FUNCTION_BLOCK F_UINT_TO_LINT (* convert UINT to LINT *)
  (* Standard: 61131-3; Classification: type conversion function *)
  (* Version 0.0, 2011-12-25, 4DIAC-IDE, 4DIAC-Consortium *)
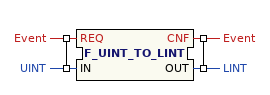
  EVENT_INPUT
    REQ WITH IN; (* Service Request *)
  END_EVENT
  EVENT_OUTPUT
    CNF WITH OUT; (* Confirmation of Requested Service *)
  END_EVENT
  VAR_INPUT
    IN : UINT; (* Event Input Qualifier *)
  END_VAR
  VAR_OUTPUT
    OUT : LINT; (* Event Output Qualifier *)
  END_VAR
END_FUNCTION_BLOCK
